(*
SPDX-FileCopyrightText: © 2026 Oleksandr Tiutyk <trofimich@gmail.com>
SPDX-License-Identifier: MIT
License: https://opensource.org/license/mit
*)

(*!
<summary>Defines an activity that waits for a configured time interval before completing.</summary>
*)

INTERFACE IDelayActivity EXTENDS IActivity

(*!
<summary>Gets or sets the total active duration, excluding time spent suspended.</summary>
<description>
Suspension retains elapsed active time. Resume waits for the remainder; a fresh start after reset
uses the full interval. Changing Interval changes the active-time target on the next running observation.
</description>
*)
{attribute 'monitoring' := 'call'}
PROPERTY Interval : TIME
GET
END_GET
SET
END_SET
END_PROPERTY

END_INTERFACE

(* stored: Version 1.1.0.1
   Itf IDelayActivity: Id {856e7c2a-9dc3-465e-921c-d949d6b76f07}
   Property Interval: Id {3c1927d5-5d68-420e-a76f-7b2f88877710}
   Get Get: Id {45b8f420-8ef4-4091-b030-9f5c0d1f7322}
   Set Set: Id {5b93a81e-24c2-437b-a101-73c188f64289} *)
